TYPE ST_BatchTrail :
STRUCT
	Batch				:STRING(100);
	Event				:STRING(100);
	Description			:STRING(100);
	User				:STRING(100);
	Oldvalue			:STRING(100);
	Newvalue			:STRING(100);
END_STRUCT
END_TYPE

(* stored: Version 1.1.0.1, ProductVersion 3.1.4026.13
   DUT ST_BatchTrail: Id {bf09939b-a695-4069-956a-45b23dc08361} *)
